INTERFACE ITF_Group3_HMI_Init EXTENDS ITF_BaseGroupElement, ITF_Group3_HMI_Connector

END_INTERFACE

(* stored: Version 1.1.0.1
   Itf ITF_Group3_HMI_Init: Id {128eddf9-5b05-0a45-2010-6a416c28c8a3} *)
